DATA_BLOCK DB 107
TITLE =
VERSION : 0.0

 FB 107
BEGIN

modes.WKM1PROC.auto := TRUE;

END_DATA_BLOCK